// TIA Portal V18 export
DATA_BLOCK "Station1LoadData"   // DB510
{ S7_Optimized_Access := 'FALSE' }
// stored: AutoNumber false
   VAR
      "PLC.PartTypeID" : Int;
      "PLC.Station1RecipeNo" : Int;
      "PLC.Station1DMXCode" : String[128];
      "PLC.StationStatus" : Int;
      "MES.ErrorCode" : Int;
      "MES.StatusBits" : DInt;
      "MES.Cycle_ID" : DInt;
      "MES.Unit_ParttypeID" : Int;
   END_VAR
BEGIN
END_DATA_BLOCK
